Staubli VAL3: strfillchr.pgx

public program strfillchr(string pStrIn, string& pStrOut[], string pChar)
  local num lIndex
begin
  //---------------------------------
  //  F I L L   O N E   S T R I N G
  //---------------------------------
  // To fill the string with custom
  // character
  //
  //
  pStrOut=""
  if getDisplayLen(pStrIn)>0
    for lIndex=0 to (getDisplayLen(pStrIn)-1)
      pStrOut=pStrOut+pChar
    endFor
  endIf
end
